Yaskawa INFORM job: KRIS7(1)_V2.JBI

/JOB
//NAME KRIS7(1)_V2
//POS
///NPOS 133,133,133,13,0,0
///TOOL 0
///POSTYPE PULSE
///PULSE
C00000=27820,-86440,-90587,-9957,54088,76092
C00001=3271,-119374,-120746,-350,28955,423
C00002=-140235,-154096,-123138,2898,12995,-682
C00003=-200060,-156091,-101839,15852,59862,-55345
C00004=-81018,-22368,15352,11535,43694,-10760
C00005=-82220,-12770,25334,12334,42674,-11455
C00006=-82220,-11619,27495,12508,41954,-11560
C00007=-82220,-11847,27069,12473,42095,-11540
C00008=-82921,-9583,28807,12754,42287,-11838
C00009=-82839,-9854,28597,12721,42264,-11802
C00010=-82839,-10288,27783,12653,42536,-11762
C00011=-82987,-9794,28166,12713,42576,-11825
C00012=-82987,-9519,28676,12758,42403,-11847
C00013=-82987,-9667,28396,12734,42496,-11833
C00014=-83090,-9325,28661,12774,42522,-11877
C00015=-82753,-11045,26659,12547,42813,-11678
C00016=-119816,-37733,5380,24735,50291,-26788
C00017=-118732,-28444,14282,24759,49358,-26561
C00018=-118732,-27369,16233,24992,48768,-26724
C00019=-118733,-27539,15928,24955,48860,-26698
C00020=-118781,-24844,17728,24865,49124,-26646
C00021=-118771,-25424,17338,24885,49069,-26656
C00022=-118771,-25846,16569,24792,49302,-26592
C00023=-118785,-25058,17100,24768,49376,-26577
C00024=-118785,-24858,17464,24811,49265,-26606
C00025=-118785,-24952,17291,24791,49318,-26592
C00026=-118793,-24494,17602,24777,49360,-26584
C00027=-118763,-26610,15508,24704,49533,-26524
C00028=-155285,-26516,12514,28456,62214,-38311
C00029=-152438,-18325,21238,28659,60298,-37701
C00030=-152440,-17188,23354,28851,59667,-37879
C00031=-152440,-17414,22937,28813,59790,-37845
C00032=-151830,-15112,24623,28749,59726,-37617
C00033=-151901,-15387,24419,28758,59733,-37642
C00034=-151901,-15814,23624,28683,59971,-37576
C00035=-151771,-15314,23995,28670,59956,-37527
C00036=-151769,-15045,24491,28721,59807,-37565
C00037=-151767,-15191,24216,28696,59889,-37542
C00038=-151679,-14843,24474,28688,59877,-37510
C00039=-151971,-16573,22523,28616,60244,-37525
C00040=-150216,-29821,9901,28279,60539,-36735
C00041=-129415,-40611,3678,-20754,45854,21846
C00042=-132229,-30881,12703,-20034,44681,20835
C00043=-132233,-29758,14737,-20264,44044,20982
C00044=-132233,-29979,14337,-20217,44170,20950
C00045=-131980,-27625,15872,-20209,44476,20997
C00046=-132007,-27902,15689,-20213,44443,20995
C00047=-132009,-28325,14925,-20124,44681,20937
C00048=-131956,-27813,15263,-20122,44745,20946
C00049=-131946,-27551,15737,-20184,44594,20990
C00050=-131944,-27692,15476,-20156,44679,20973
C00051=-131906,-27334,15713,-20158,44724,20979
C00052=-132026,-29082,13878,-20039,44914,20879
C00053=-163713,-23600,14498,-6442,42405,6672
C00054=-163955,-12441,25582,-6447,41301,6644
C00055=-163960,-11291,27745,-6536,40565,6698
C00056=-163959,-11518,27319,-6518,40711,6685
C00057=-163182,-9327,29005,-6883,40857,7042
C00058=-163270,-9587,28803,-6845,40841,7005
C00059=-163272,-10021,27989,-6806,41118,6980
C00060=-163107,-9544,28360,-6883,41148,7055
C00061=-163099,-9280,28861,-6910,40971,7077
C00062=-163096,-9426,28582,-6901,41068,7072
C00063=-162981,-9093,28842,-6958,41088,7124
C00064=-163354,-10779,26863,-6731,41408,6921
C00065=-188135,19294,49745,5326,42598,-4607
C00066=-187094,34022,67542,5190,39163,-4331
C00067=-187099,35860,70809,5317,38103,-4403
C00068=-187098,35492,70157,5290,38315,-4390
C00069=-186242,38033,72879,4886,37897,-3996
C00070=-186340,37725,72546,4929,37948,-4039
C00071=-186342,37004,71278,4886,38357,-4015
C00072=-186159,37561,71878,4800,38266,-3932
C00073=-186153,37998,72654,4828,38007,-3942
C00074=-186151,37748,72215,4808,38149,-3930
C00075=-186023,38140,72638,4745,38082,-3873
C00076=-186437,35890,69530,4881,38858,-4029
C00077=-129415,-40611,3678,-20754,45854,21846
C00078=-138780,-33942,5724,-2673,47750,14957
C00079=-138299,-28740,11900,-2889,46638,15192
C00080=-170916,-2374,31381,8191,49243,1565
C00081=-171700,-5880,26786,8312,50334,1335
C00082=-135165,-49074,-6503,-3925,47635,16482
C00083=-161317,-13185,16777,20608,75826,-36642
C00084=-161248,734,29994,20695,74889,-36781
C00085=-160775,4102,35532,20888,73203,-36913
C00086=-160685,10042,42080,20996,72268,-37049
C00087=-152044,455,33682,21552,70401,-34333
C00088=-119342,-11696,23952,21569,62028,-23940
C00089=-119305,-17523,16883,21319,63284,-23678
C00090=-135165,-49074,-6503,-3925,47635,16482
C00091=-129415,-40611,3678,-20754,45854,21846
C00092=-171396,-8104,23990,8148,50880,1508
C00093=-171152,-2065,31577,8260,49305,1472
C00094=-192271,67900,104631,16357,43373,-8337
C00095=-192892,57382,88980,15390,47553,-7857
C00096=-135165,-49074,-6503,-3925,47635,16482
C00097=-161317,-13185,16777,20608,75826,-36642
C00098=-119244,-24750,9342,21153,64138,-23490
C00099=-119300,-17410,17676,21394,62882,-23755
C00100=-119343,-11696,23952,21569,62027,-23940
C00101=-84728,5286,37848,17156,54382,-11867
C00102=-85414,851,32833,17125,55288,-11988
C00103=-135165,-49074,-6503,-3925,47635,16482
C00104=-129360,-40332,3441,-20673,46138,21804
C00105=-138676,-33640,5524,-2697,48031,14993
C00106=-138191,-28354,11811,-2916,46896,15229
C00107=-170671,-2058,31280,8087,49442,1685
C00108=-171477,-5655,26582,8215,50551,1445
C00109=-135070,-48777,-6734,-3939,47933,16510
C00110=-161130,-12883,16630,20602,76011,-36544
C00111=-158859,-1544,27720,20849,74530,-36001
C00112=-160132,3814,34899,20915,73276,-36675
C00113=-163971,-71,35306,26985,66016,-40466
C00114=-154970,-9958,27505,27337,62784,-37857
C00115=-119242,-19669,19375,23179,54823,-25430
C00116=-119312,-17166,16760,21274,63528,-23633
C00117=-135070,-48777,-6734,-3939,47933,16510
C00118=-129360,-40332,3441,-20673,46138,21804
C00119=-171172,-7872,23791,8052,51098,1618
C00120=-170796,-1768,31531,8129,49447,1635
C00121=-191948,67436,103535,16137,43742,-8121
C00122=-192674,57393,88583,15275,47758,-7731
C00123=-135070,-48777,-6734,-3939,47933,16510
C00124=-161130,-12883,16630,20602,76011,-36544
C00125=-119252,-24388,9211,21109,64389,-23445
C00126=-119307,-17059,17547,21348,63127,-23710
C00127=-115642,-27884,15061,20579,45940,-25049
C00128=-76385,-6634,29757,2420,43140,-7452
C00129=-85568,1158,32706,17108,55544,-12007
C00130=-135070,-48777,-6734,-3939,47933,16510
C00131=-134221,-121505,-102040,30238,34212,-41263
C00132=3271,-119374,-120746,-350,28955,423
BC00000=193141,673698,861874
BC00001=132383,666204,1075229
BC00002=261940,799209,1050994
BC00003=248524,1011966,1050994
BC00004=257490,879918,1075175
BC00005=257490,892976,975703
BC00006=257490,892976,975703
BC00007=257490,892976,975703
BC00008=257490,892976,975703
BC00009=257490,892976,975703
BC00010=257490,892976,975703
BC00011=257490,892976,975703
BC00012=257490,892976,975703
BC00013=257490,892976,975703
BC00014=257490,892976,975703
BC00015=257490,892976,975703
BC00016=257490,892975,975706
BC00017=257490,892976,975703
BC00018=257490,892976,975703
BC00019=257490,892976,975703
BC00020=257490,892976,975703
BC00021=257490,892976,975703
BC00022=257490,892976,975703
BC00023=257490,892976,975703
BC00024=257490,892976,975703
BC00025=257490,892976,975703
BC00026=257490,892976,975703
BC00027=257490,892976,975703
BC00028=257490,892975,975706
BC00029=257490,892976,975703
BC00030=257490,892976,975703
BC00031=257490,892976,975703
BC00032=257490,892976,975703
BC00033=257490,892976,975703
BC00034=257490,892976,975703
BC00035=257490,892976,975703
BC00036=257490,892976,975703
BC00037=257490,892976,975703
BC00038=257490,892976,975703
BC00039=257490,892976,975703
BC00040=257490,892976,975703
BC00041=257490,892975,975706
BC00042=257490,892976,975703
BC00043=257490,892976,975703
BC00044=257490,892976,975703
BC00045=257490,892976,975703
BC00046=257490,892976,975703
BC00047=257490,892976,975703
BC00048=257490,892976,975703
BC00049=257490,892976,975703
BC00050=257490,892976,975703
BC00051=257490,892976,975703
BC00052=257490,892976,975703
BC00053=257490,892975,975706
BC00054=257490,892976,975703
BC00055=257490,892976,975703
BC00056=257490,892976,975703
BC00057=257490,892976,975703
BC00058=257490,892976,975703
BC00059=257490,892976,975703
BC00060=257490,892976,975703
BC00061=257490,892976,975703
BC00062=257490,892976,975703
BC00063=257490,892976,975703
BC00064=257490,892976,975703
BC00065=257490,892975,975706
BC00066=257490,892976,975703
BC00067=257490,892976,975703
BC00068=257490,892976,975703
BC00069=257490,892976,975703
BC00070=257490,892976,975703
BC00071=257490,892976,975703
BC00072=257490,892976,975703
BC00073=257490,892976,975703
BC00074=257490,892976,975703
BC00075=257490,892976,975703
BC00076=257490,892976,975703
BC00077=257490,892975,975706
BC00078=257490,892976,975703
BC00079=257490,892976,975703
BC00080=257490,892976,975703
BC00081=257490,892976,975703
BC00082=257490,892976,975703
BC00083=257490,892976,975703
BC00084=257490,892976,975703
BC00085=257490,892976,975703
BC00086=257490,892976,975703
BC00087=257490,892976,975703
BC00088=257490,892976,975703
BC00089=257490,892976,975703
BC00090=257490,892976,975703
BC00091=257490,892975,975706
BC00092=257490,892976,975703
BC00093=257490,892976,975703
BC00094=257490,892976,975703
BC00095=257490,892976,975703
BC00096=257490,892976,975703
BC00097=257490,892976,975703
BC00098=257490,892976,975703
BC00099=257490,892976,975703
BC00100=257490,892976,975703
BC00101=257490,892976,975703
BC00102=257490,892976,975703
BC00103=257490,892976,975703
BC00104=257490,892975,975706
BC00105=257490,892976,975703
BC00106=257490,892976,975703
BC00107=257490,892976,975703
BC00108=257490,892976,975703
BC00109=257490,892976,975703
BC00110=257490,892976,975703
BC00111=257490,892976,975703
BC00112=257490,892976,975703
BC00113=257490,892976,975703
BC00114=257490,892976,975703
BC00115=257490,892976,975703
BC00116=257490,892976,975703
BC00117=257490,892976,975703
BC00118=257490,892975,975706
BC00119=257490,892976,975703
BC00120=257490,892976,975703
BC00121=257490,892976,975702
BC00122=257490,892976,975703
BC00123=257490,892976,975703
BC00124=257490,892976,975703
BC00125=257490,892976,975703
BC00126=257490,892976,975703
BC00127=257490,892976,975703
BC00128=257490,892976,975703
BC00129=257490,892976,975703
BC00130=257490,892976,975703
BC00131=285803,889729,975706
BC00132=132383,679261,975760
EC00000=0,556476
EC00001=266052,556475
EC00002=487668,556475
EC00003=266052,556475
EC00004=492425,556475
EC00005=492424,556474
EC00006=492424,556474
EC00007=492424,556474
EC00008=492424,556474
EC00009=492424,556474
EC00010=492424,556474
EC00011=492424,556474
EC00012=492424,556474
EC00013=492424,556474
EC00014=492424,556474
EC00015=492424,556474
EC00016=492425,556475
EC00017=492424,556474
EC00018=492424,556474
EC00019=492424,556474
EC00020=492424,556474
EC00021=492424,556474
EC00022=492424,556474
EC00023=492424,556474
EC00024=492424,556474
EC00025=492424,556474
EC00026=492424,556474
EC00027=492424,556474
EC00028=492425,556475
EC00029=492424,556474
EC00030=492424,556474
EC00031=492424,556474
EC00032=492424,556474
EC00033=492424,556474
EC00034=492424,556474
EC00035=492424,556474
EC00036=492424,556474
EC00037=492424,556474
EC00038=492424,556474
EC00039=492424,556474
EC00040=492424,556474
EC00041=492425,556475
EC00042=492424,556474
EC00043=492424,556474
EC00044=492424,556474
EC00045=492424,556474
EC00046=492424,556474
EC00047=492424,556474
EC00048=492424,556474
EC00049=492424,556474
EC00050=492424,556474
EC00051=492424,556474
EC00052=492424,556474
EC00053=492425,556475
EC00054=492424,556474
EC00055=492424,556474
EC00056=492424,556474
EC00057=492424,556474
EC00058=492424,556474
EC00059=492424,556474
EC00060=492424,556474
EC00061=492424,556474
EC00062=492424,556474
EC00063=492424,556474
EC00064=492424,556474
EC00065=492425,556475
EC00066=492424,556474
EC00067=492424,556474
EC00068=492424,556474
EC00069=492424,556474
EC00070=492424,556474
EC00071=492424,556474
EC00072=492424,556474
EC00073=492424,556474
EC00074=492424,556474
EC00075=492424,556474
EC00076=492424,556474
EC00077=492425,556475
EC00078=492424,556474
EC00079=492424,556474
EC00080=492424,556474
EC00081=492424,556474
EC00082=492424,556474
EC00083=492424,556474
EC00084=492424,556474
EC00085=492424,556474
EC00086=492424,556474
EC00087=492424,556474
EC00088=492424,556474
EC00089=492424,556474
EC00090=492424,556474
EC00091=492425,556475
EC00092=492424,556474
EC00093=492424,556474
EC00094=492424,556474
EC00095=492424,556474
EC00096=492424,556474
EC00097=492424,556474
EC00098=492424,556474
EC00099=492424,556474
EC00100=492424,556474
EC00101=492424,556474
EC00102=492424,556474
EC00103=492424,556474
EC00104=492425,556475
EC00105=492424,556474
EC00106=492424,556474
EC00107=492424,556474
EC00108=492424,556474
EC00109=492424,556474
EC00110=492424,556474
EC00111=492424,556474
EC00112=492424,556474
EC00113=492424,556474
EC00114=492424,556474
EC00115=492424,556474
EC00116=492424,556474
EC00117=492424,556474
EC00118=492425,556475
EC00119=492424,556474
EC00120=492424,556474
EC00121=492423,556474
EC00122=492424,556474
EC00123=492424,556474
EC00124=492424,556474
EC00125=492424,556474
EC00126=492424,556474
EC00127=492424,556474
EC00128=492424,556474
EC00129=492424,556474
EC00130=492424,556474
EC00131=443420,556475
EC00132=443420,556475
///POSTYPE BASE
///RECTAN
///RCONF 0,0,0,0,0,0,0,0,0,0,0,0,0,0,0,0,0,0,0,0,0,0,0,0
P00006=0.222,-3.123,-1.508,0.0000,0.0000,0.0000
P00040=-0.030,9.648,2.467,0.0000,0.0000,0.0000
P00041=0.192,3.924,0.305,0.0000,0.0000,0.0000
P00042=-0.217,1.941,0.413,0.0000,0.0000,0.0000
P00043=-0.044,-1.937,1.197,0.0000,0.0000,0.0000
P00044=0.687,-2.322,1.156,0.0000,0.0000,0.0000
P00045=-0.068,-0.810,1.603,0.0000,0.0000,0.0000
P00050=4.296,-4.501,-0.826,0.0000,0.0000,0.0000
P00051=0.367,3.892,0.009,0.0000,0.0000,0.0000
P00052=0.088,2.832,-0.342,0.0000,0.0000,0.0000
P00053=0.134,6.594,0.107,0.0000,0.0000,0.0000
P00054=-0.103,6.509,-0.702,0.0000,0.0000,0.0000
P00055=-0.342,8.912,1.324,0.0000,0.0000,0.0000
//INST
///DATE 2025/05/21 08:28
///ATTR SC,RW
///GROUP1 RB1,BS1
///GROUP2 ST1
NOP
CALL JOB:CLEAN-R1_KM_3P
MOVJ C00000 BC00000 VJ=100.00  +MOVJ EC00000 VJ=100.00
MOVJ C00001 BC00001 VJ=100.00  +MOVJ EC00001 VJ=100.00
MOVJ C00002 BC00002 VJ=100.00  +MOVJ EC00002 VJ=100.00
MOVJ C00003 BC00003 VJ=100.00  +MOVJ EC00003 VJ=100.00
SFTOF3D
MOVL C00004 BC00004 V=666.7  +MOVJ EC00004 VJ=100.00
SMOVL C00005 BC00005 V=166.7  +MOVJ EC00005
SREFP 3 C00006 BC00006  +REFP EC00006
CALL JOB:SEARCH-R1-S13D
SET P041 P006
SFTON3D P041
SMOVL C00007 BC00007 V=166.7  +MOVJ EC00007
SREFP 3 C00008 BC00008  +REFP EC00008
CALL JOB:SEARCH-R1-S13D
SET P041 P006
SFTON3D P041
SMOVL C00009 BC00009 V=166.7  +MOVJ EC00009
SMOVL C00010 BC00010 V=166.7  +MOVJ EC00010
SMOVL C00011 BC00011 V=166.7  +MOVJ EC00011
SREFP 3 C00012 BC00012  +REFP EC00012
CALL JOB:SEARCH-R1-S13D
SET P051 P006
SFTON3D P051
SMOVL C00013 BC00013 V=100.0  +MOVJ EC00013
SREFP 3 C00014 BC00014  +REFP EC00014
CALL JOB:SEARCH-R1-S13D
SET P051 P006
SFTON3D P051
SMOVL C00015 BC00015 V=166.7  +MOVJ EC00015
SFTOF3D
MOVL C00016 BC00016 V=666.7  +MOVJ EC00016 VJ=100.00
SMOVL C00017 BC00017 V=166.7  +MOVJ EC00017
SREFP 3 C00018 BC00018  +REFP EC00018
CALL JOB:SEARCH-R1-S13D
SET P042 P006
SFTON3D P042
SMOVL C00019 BC00019 V=166.7  +MOVJ EC00019
SREFP 3 C00020 BC00020  +REFP EC00020
CALL JOB:SEARCH-R1-S13D
SET P042 P006
SFTON3D P042
SMOVL C00021 BC00021 V=166.7  +MOVJ EC00021
SMOVL C00022 BC00022 V=166.7  +MOVJ EC00022
SMOVL C00023 BC00023 V=166.7  +MOVJ EC00023
SREFP 3 C00024 BC00024  +REFP EC00024
CALL JOB:SEARCH-R1-S13D
SET P052 P006
SFTON3D P052
SMOVL C00025 BC00025 V=100.0  +MOVJ EC00025
SREFP 3 C00026 BC00026  +REFP EC00026
CALL JOB:SEARCH-R1-S13D
SET P052 P006
SFTON3D P052
SMOVL C00027 BC00027 V=166.7  +MOVJ EC00027
SFTOF3D
MOVL C00028 BC00028 V=666.7  +MOVJ EC00028 VJ=100.00
SMOVL C00029 BC00029 V=166.7  +MOVJ EC00029
SREFP 3 C00030 BC00030  +REFP EC00030
CALL JOB:SEARCH-R1-S13D
SET P043 P006
SFTON3D P043
SMOVL C00031 BC00031 V=166.7  +MOVJ EC00031
SREFP 3 C00032 BC00032  +REFP EC00032
CALL JOB:SEARCH-R1-S13D
SET P043 P006
SFTON3D P043
SMOVL C00033 BC00033 V=166.7  +MOVJ EC00033
SMOVL C00034 BC00034 V=166.7  +MOVJ EC00034
SMOVL C00035 BC00035 V=166.7  +MOVJ EC00035
SREFP 3 C00036 BC00036  +REFP EC00036
CALL JOB:SEARCH-R1-S13D
SET P053 P006
SFTON3D P053
SMOVL C00037 BC00037 V=100.0  +MOVJ EC00037
SREFP 3 C00038 BC00038  +REFP EC00038
CALL JOB:SEARCH-R1-S13D
SET P053 P006
SFTON3D P053
SMOVL C00039 BC00039 V=166.7  +MOVJ EC00039
SFTOF3D
MOVL C00040 BC00040 V=666.7  +MOVJ EC00040 VJ=100.00
MOVL C00041 BC00041 V=666.7  +MOVJ EC00041 VJ=100.00
SMOVL C00042 BC00042 V=166.7  +MOVJ EC00042
SREFP 3 C00043 BC00043  +REFP EC00043
CALL JOB:SEARCH-R1-S13D
SET P044 P006
SFTON3D P044
SMOVL C00044 BC00044 V=166.7  +MOVJ EC00044
SREFP 3 C00045 BC00045  +REFP EC00045
CALL JOB:SEARCH-R1-S13D
SET P044 P006
SFTON3D P044
SMOVL C00046 BC00046 V=166.7  +MOVJ EC00046
SMOVL C00047 BC00047 V=166.7  +MOVJ EC00047
SMOVL C00048 BC00048 V=166.7  +MOVJ EC00048
SREFP 3 C00049 BC00049  +REFP EC00049
CALL JOB:SEARCH-R1-S13D
SET P054 P006
SFTON3D P054
SMOVL C00050 BC00050 V=100.0  +MOVJ EC00050
SREFP 3 C00051 BC00051  +REFP EC00051
CALL JOB:SEARCH-R1-S13D
SET P054 P006
SFTON3D P054
SMOVL C00052 BC00052 V=166.7  +MOVJ EC00052
SFTOF3D
MOVL C00053 BC00053 V=666.7  +MOVJ EC00053 VJ=100.00
SMOVL C00054 BC00054 V=166.7  +MOVJ EC00054
SREFP 3 C00055 BC00055  +REFP EC00055
CALL JOB:SEARCH-R1-S13D
SET P045 P006
SFTON3D P045
SMOVL C00056 BC00056 V=166.7  +MOVJ EC00056
SREFP 3 C00057 BC00057  +REFP EC00057
CALL JOB:SEARCH-R1-S13D
SET P045 P006
SFTON3D P045
SMOVL C00058 BC00058 V=166.7  +MOVJ EC00058
SMOVL C00059 BC00059 V=166.7  +MOVJ EC00059
SMOVL C00060 BC00060 V=166.7  +MOVJ EC00060
SREFP 3 C00061 BC00061  +REFP EC00061
CALL JOB:SEARCH-R1-S13D
SET P055 P006
SFTON3D P055
SMOVL C00062 BC00062 V=100.0  +MOVJ EC00062
SREFP 3 C00063 BC00063  +REFP EC00063
CALL JOB:SEARCH-R1-S13D
SET P055 P006
SFTON3D P055
SMOVL C00064 BC00064 V=166.7  +MOVJ EC00064
SFTOF3D
MOVL C00065 BC00065 V=666.7  +MOVJ EC00065 VJ=100.00
SMOVL C00066 BC00066 V=166.7  +MOVJ EC00066
SREFP 3 C00067 BC00067  +REFP EC00067
CALL JOB:SEARCH-R1-S13D
SET P040 P006
SFTON3D P040
SMOVL C00068 BC00068 V=166.7  +MOVJ EC00068
SREFP 3 C00069 BC00069  +REFP EC00069
CALL JOB:SEARCH-R1-S13D
SET P040 P006
SFTON3D P040
SMOVL C00070 BC00070 V=166.7  +MOVJ EC00070
SMOVL C00071 BC00071 V=166.7  +MOVJ EC00071
SMOVL C00072 BC00072 V=166.7  +MOVJ EC00072
SREFP 3 C00073 BC00073  +REFP EC00073
CALL JOB:SEARCH-R1-S13D
SET P050 P006
SFTON3D P050
SMOVL C00074 BC00074 V=100.0  +MOVJ EC00074
SREFP 3 C00075 BC00075  +REFP EC00075
CALL JOB:SEARCH-R1-S13D
SET P050 P006
SFTON3D P050
SMOVL C00076 BC00076 V=166.7  +MOVJ EC00076
SFTOF3D
MOVL C00077 BC00077 V=666.7  +MOVJ EC00077 VJ=100.00
SFTON3D P044
SMOVL C00078 BC00078 V=166.7  +MOVJ EC00078
SMOVL C00079 BC00079 V=166.7 PL=0  +MOVJ EC00079
MACRO1 MJ#(0) ARGF9
ARCON
SFTON3D P045
SMOVL C00080 BC00080 V=10.8  +MOVJ EC00080
ARCOF
MOVL C00081 BC00081 V=166.7  +MOVJ EC00081 VJ=100.00
SFTOF3D
SMOVL C00082 BC00082 V=666.7  +MOVJ EC00082
SMOVL C00083 BC00083 V=666.7  +MOVJ EC00083
MOVL C00084 BC00084 V=666.7  +MOVJ EC00084 VJ=100.00
SFTON3D P044
SMOVL C00085 BC00085 V=166.7  +MOVJ EC00085
SMOVL C00086 BC00086 V=166.7 PL=0  +MOVJ EC00086
MACRO1 MJ#(0) ARGF9
ARCON
SFTON3D P043
SMOVL C00087 BC00087 V=10.8  +MOVJ EC00087
SFTON3D P042
SMOVL C00088 BC00088 V=10.8  +MOVJ EC00088
ARCOF
MOVL C00089 BC00089 V=166.7  +MOVJ EC00089 VJ=100.00
SFTOF3D
SMOVL C00090 BC00090 V=666.7  +MOVJ EC00090
SFTOF3D
MOVL C00091 BC00091 V=666.7  +MOVJ EC00091 VJ=100.00
SFTON3D P045
SMOVL C00092 BC00092 V=166.7  +MOVJ EC00092
SMOVL C00093 BC00093 V=166.7 PL=0  +MOVJ EC00093
MACRO1 MJ#(0) ARGF9
ARCON
SFTON3D P040
SMOVL C00094 BC00094 V=10.8  +MOVJ EC00094
ARCOF
MOVL C00095 BC00095 V=166.7  +MOVJ EC00095 VJ=100.00
SFTOF3D
SMOVL C00096 BC00096 V=666.7  +MOVJ EC00096
SMOVL C00097 BC00097 V=666.7  +MOVJ EC00097
MOVL C00098 BC00098 V=666.7  +MOVJ EC00098 VJ=100.00
SFTON3D P042
SMOVL C00099 BC00099 V=166.7  +MOVJ EC00099
SMOVL C00100 BC00100 V=166.7 PL=0  +MOVJ EC00100
MACRO1 MJ#(0) ARGF9
ARCON
SFTON3D P041
SMOVL C00101 BC00101 V=10.8  +MOVJ EC00101
ARCOF
MOVL C00102 BC00102 V=166.7  +MOVJ EC00102 VJ=100.00
SFTOF3D
SMOVL C00103 BC00103 V=666.7  +MOVJ EC00103
MOVL C00104 BC00104 V=666.7  +MOVJ EC00104 VJ=100.00
SFTON3D P054
SMOVL C00105 BC00105 V=166.7  +MOVJ EC00105
SMOVL C00106 BC00106 V=166.7 PL=0  +MOVJ EC00106
MACRO1 MJ#(0) ARGF9
ARCON
SFTON3D P055
SMOVL C00107 BC00107 V=10.0  +MOVJ EC00107
ARCOF
MOVL C00108 BC00108 V=166.7  +MOVJ EC00108 VJ=100.00
SFTOF3D
SMOVL C00109 BC00109 V=666.7  +MOVJ EC00109
SMOVL C00110 BC00110 V=666.7  +MOVJ EC00110
MOVL C00111 BC00111 V=666.7  +MOVJ EC00111 VJ=100.00
SFTON3D P054
SMOVL C00112 BC00112 V=166.7  +MOVJ EC00112
SMOVL C00113 BC00113 V=166.7 PL=0  +MOVJ EC00113
MACRO1 MJ#(0) ARGF9
ARCON
SFTON3D P053
SMOVL C00114 BC00114 V=10.0  +MOVJ EC00114
SFTON3D P052
SMOVL C00115 BC00115 V=10.0  +MOVJ EC00115
ARCOF
MOVL C00116 BC00116 V=166.7  +MOVJ EC00116 VJ=100.00
SFTOF3D
SMOVL C00117 BC00117 V=666.7  +MOVJ EC00117
SFTOF3D
MOVL C00118 BC00118 V=666.7  +MOVJ EC00118 VJ=100.00
SFTON3D P055
SMOVL C00119 BC00119 V=166.7  +MOVJ EC00119
SMOVL C00120 BC00120 V=166.7 PL=0  +MOVJ EC00120
MACRO1 MJ#(0) ARGF9
ARCON
SFTON3D P050
SMOVL C00121 BC00121 V=10.0  +MOVJ EC00121
ARCOF
MOVL C00122 BC00122 V=166.7  +MOVJ EC00122 VJ=100.00
SFTOF3D
SMOVL C00123 BC00123 V=666.7  +MOVJ EC00123
SMOVL C00124 BC00124 V=666.7  +MOVJ EC00124
MOVL C00125 BC00125 V=666.7  +MOVJ EC00125 VJ=100.00
SFTON3D P052
SMOVL C00126 BC00126 V=166.7  +MOVJ EC00126
SMOVL C00127 BC00127 V=166.7 PL=0  +MOVJ EC00127
MACRO1 MJ#(0) ARGF9
ARCON
SFTON3D P051
SMOVL C00128 BC00128 V=10.0  +MOVJ EC00128
ARCOF
MOVL C00129 BC00129 V=166.7  +MOVJ EC00129 VJ=100.00
SFTOF3D
SMOVL C00130 BC00130 V=666.7  +MOVJ EC00130
MOVJ C00131 BC00131 VJ=100.00  +MOVJ EC00131 VJ=100.00
'
'
'
MOVJ C00132 BC00132 VJ=100.00  +MOVJ EC00132 VJ=100.00
END
